// Brief: Master Arm Initialization
FUNCTION_BLOCK PUBLIC FB_ArmClutch EXTENDS FB_MasterArmCtrlBase
VAR_INPUT
END_VAR
VAR_OUTPUT
END_VAR
VAR
END_VAR

END_FUNCTION_BLOCK

(* stored: Version 1.1.0.1, ProductVersion 3.1.4024.12
   POU FB_ArmClutch: Id {093bd9ec-6cc6-4389-91e4-f8586e50bb1f}, SpecialFunc None *)
